// TIA Portal V19 export
TYPE "typeFDoorFunction"
// Safety status of door
// stored: Access Published, IsFailsafeCompliant true, Namespace Safety
   STRUCT
      released { ExternalWritable := 'False'} : Bool;   // Door OK
      ackReq { ExternalWritable := 'False'} : Bool;   // Acknowledge required
   END_STRUCT;
END_TYPE
